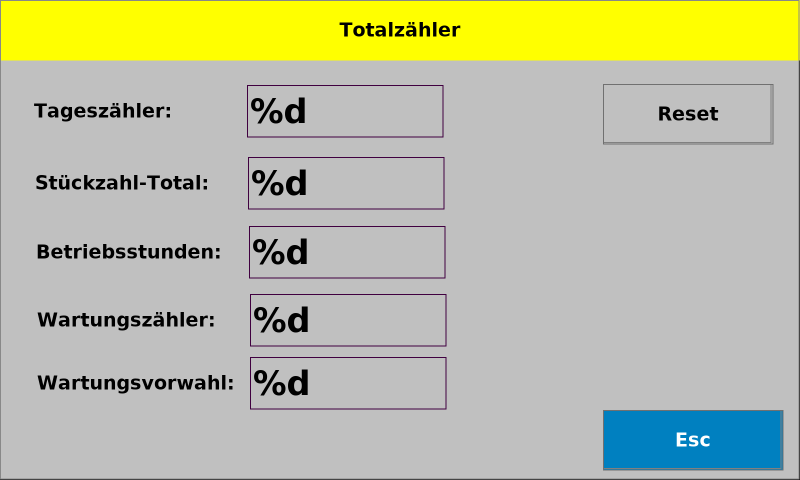
VISUALIZATION Total  // 800x480
    Rectangle (0,0 800x480)
    Rectangle (0,0 800x60), "Totalzähler"
    Button (603,410 180x60), "Esc"
        OnMouseUp: change screen: Previous 
    Rectangle (247,85 196x52), "%d", text variable: DB6.diTagesZaehler
    Label (31,94 208x34), "Tageszähler:"
    Rectangle (248,157 196x52), "%d", text variable: DB6.diStueck_Total
    Label (32,166 209x34), "Stückzahl-Total:"
    Button (603,84 170x60), "Reset"
    Rectangle (249,226 196x52), "%d", text variable: DB6.runTime.hours
    Label (33,235 209x34), "Betriebsstunden:"
    Rectangle (250,294 196x52), "%d", text variable: DB6.diReinigung_Zaehl
    Label (34,303 209x34), "Wartungszähler:"
    Label (34,366 209x34), "Wartungsvorwahl:"
    Rectangle (250,357 196x52), "%d", text variable: DB6.diReinigung_Vorw
END_VISUALIZATION

(* stored: Version 1.1.0.1, ProductVersion 3.1.4024.3
   Visu Total: Id {6dbeb29c-85e0-4c16-8c76-a7030040116d} *)
